FUNCTION_BLOCK FB_AcceptTCP
VAR_INPUT
END_VAR
VAR_OUTPUT
END_VAR
VAR
END_VAR

METHOD PUBLIC M_SocketAccept
VAR_INPUT
END_VAR
END_METHOD

METHOD PUBLIC M_SocketListen
VAR_INPUT
END_VAR
END_METHOD

END_FUNCTION_BLOCK

(* stored: Version 1.1.0.1, ProductVersion 3.1.4024.12
   POU FB_AcceptTCP: Id {689663a5-455a-48ee-a140-0c6ca4007826}, SpecialFunc None
   Method M_SocketAccept: Id {20c1851f-05ee-4536-98d4-083ac4e68a01}
   Method M_SocketListen: Id {66c732dc-ca30-4c0e-b95f-3a2e2248d25d} *)
